// TIA Portal V17 export
// export: Created 2023-02-14T02:49:22.1667963Z, ExportSetting WithDefaults, DisplayName Totally Integrated Automation Portal, DisplayVersion V17, DisplayName TIA Portal Openness, DisplayVersion V17, DisplayName TIA Portal Teamcenter Gateway, DisplayVersion V17, DisplayName TIA Portal Version Control Interface, DisplayVersion V17, DisplayName SINAMICS Startdrive Advanced, DisplayVersion V17, DisplayName SINAMICS Startdrive G130, G150, S120, S150, SINAMICS MV, S210, DisplayVersion V17, DisplayName SINAMICS Startdrive G110M, G120, G120C, G120D, G120P, G115D, DisplayVersion V17, DisplayName STEP 7 Professional, DisplayVersion V17, DisplayName STEP 7 Safety, DisplayVersion V17, DisplayName WinCC Professional, DisplayVersion V17
DATA_BLOCK "IO Motor MCC Panel Blending_DB"   // DB5
VERSION : 0.1
// stored: AutoNumber true, DBAccessibleFromOPCUA true, DBAccessibleFromWebserver true, InstanceOfName IO Motor MCC Panel Blending, InstanceOfType FB
"IO Motor MCC Panel Blending"
   // VAR_INPUT
   //    lock : Bool;
   //    Init : Bool;
   //    Reset : Bool;
   // END_VAR
   // VAR
   //    "XA-12.01" { S7_SetPoint := 'True'} : "Motor_w_VSD";
   //    "XA-13.01" { S7_SetPoint := 'True'} : "Motor_w_VSD";
   //    "P-13.02" { S7_SetPoint := 'True'} : "Motor";
   //    "XA-20.00" { S7_SetPoint := 'True'} : "Motor_w_VSD";
   //    "XA-21.00" { S7_SetPoint := 'True'} : "Motor_w_VSD";
   //    "P-21.01" { S7_SetPoint := 'True'} : "Motor_w_VSD";
   //    "P-22.01" { S7_SetPoint := 'True'} : "Motor_w_VSD";
   //    "P-22.02" { S7_SetPoint := 'True'} : "Motor";
   //    "P-22.03" { S7_SetPoint := 'True'} : "Motor_w_VSD";
   //    "P-23.01" { S7_SetPoint := 'True'} : "Motor_w_VSD";
   //    "P-24.01" { S7_SetPoint := 'True'} : "Motor_w_VSD";
   //    "P-34.01" { S7_SetPoint := 'True'} : "Motor_w_VSD";
   //    "XA-30.00" { S7_SetPoint := 'True'} : "Motor_w_VSD";
   //    "XA-31.00" { S7_SetPoint := 'True'} : "Motor_w_VSD";
   //    "P-31.01" { S7_SetPoint := 'True'} : "Motor_w_VSD";
   //    "P-32.01" { S7_SetPoint := 'True'} : "Motor_w_VSD";
   //    "P-32.02" { S7_SetPoint := 'True'} : "Motor";
   //    "P-32.03" { S7_SetPoint := 'True'} : "Motor_w_VSD";
   //    "P-34.02" { S7_SetPoint := 'True'} : "Motor";
   //    "P-35.01" { S7_SetPoint := 'True'} : "Motor_w_VSD";
   //    "P-22_Circ" { S7_SetPoint := 'True'} : "Motor";
   //    "P-32_Circ" : "Motor";
   //    "P-81.02" { S7_SetPoint := 'True'} : "Motor";
   //    "P-81.01" { S7_SetPoint := 'True'} : "Motor_w_VSD";
   //    "P-34.01 DOL" { S7_SetPoint := 'True'} : "Motor_w_VSD";
   //    "P-84.01" { S7_SetPoint := 'True'} : "Motor_w_VSD";
   //    "P-84.02" { S7_SetPoint := 'True'} : "Motor_w_VSD";
   //    "P-82.01" { S7_SetPoint := 'True'} : "Motor_w_VSD";
   //    "XA-14.01" { S7_SetPoint := 'True'} : "Motor_w_VSD";
   //    "P-20.01" { S7_SetPoint := 'True'} : "Motor_w_VSD";
   //    "P-30.01" { S7_SetPoint := 'True'} : "Motor_w_VSD";
   //    "P-40.01" { S7_SetPoint := 'True'} : "Motor_w_VSD";
   //    "P-41.01" { S7_SetPoint := 'True'} : "Motor_w_VSD";
   //    "XA-40.00" { S7_SetPoint := 'True'} : "Motor_w_VSD";
   //    "XA-41.00" { S7_SetPoint := 'True'} : "Motor_w_VSD";
   //    "P-81.02A" { S7_SetPoint := 'True'} : "Motor";
   //    "P-24.02" { S7_SetPoint := 'True'} : "Motor";
   //    "P-82.02" { S7_SetPoint := 'True'} : "Motor";
   //    "XA-82.00" { S7_SetPoint := 'True'} : "Motor";
   //    "P-82.01A" { S7_SetPoint := 'True'} : "Motor";
   //    "P-84.01A" { S7_SetPoint := 'True'} : "Motor";
   //    "P-84.03" { S7_SetPoint := 'True'} : "Motor";
   //    "P-84.02A" { S7_SetPoint := 'True'} : "Motor";
   //    "P-84.04" { S7_SetPoint := 'True'} : "Motor";
   // END_VAR
BEGIN
   "XA-20.00".IN_SP_Speed := 5.0;
   "XA-21.00".IN_SP_Speed := 5.0;
   "P-21.01".IN_SP_Speed := 5.0;
   "XA-30.00".IN_SP_Speed := 5.0;
   "XA-31.00".IN_SP_Speed := 5.0;
   "P-31.01".IN_SP_Speed := 5.0;
   "P-32.01".IN_SP_Speed := 5.0;
   "P-32.03".IN_SP_Speed := 5.0;
END_DATA_BLOCK
